ABB RobotStudio station: w7.rspag

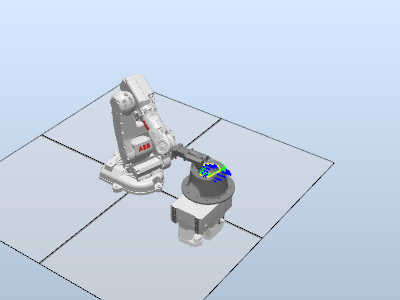
--- station ---
Station Project1 (saved by RobotStudio 22.3.10098.0)
Controller Controller1
  mechanical unit ROB_1: IRB140_6_81_C_03, 6 joints, base frame (0, 0, 0) mm
  mechanical unit M7DM1: MTD_250_M2009_REV1_01, 1 joints, base frame (584.98, -18.75, 250) mm, rotated rx 0 ry 0 rz 90 deg
Layout (positions relative to the parent item):
  - IRB140_6_81_C_03 [mechanism, from Robots\IRB140_6_81_C_G_03.rslib] at (0, 0, 0) mm; joint values [-0.3011, -0.1554, 0.7255, -0.5959, -0.6591, 0.4921] (rad or m)
  - MTD_250_M2009_REV1_01 [mechanism] at (584.98, -18.75, 250) mm, rotated rx 0 ry 0 rz 90 deg; joint values [0.0497] (rad or m)
      links: Base, Link1
  - gripped_pen [mechanism, from Components\gripped_pen.rslib] at (384.06, -95.88, 502.57) mm, rotated rx 0 ry 90 rz 2.85 deg
  - potty1 [part] at (690.16, 154.88, 241.77) mm, rotated rx 90 ry 0 rz 2.85 deg, size 275.1 x 194.8 x 257.3 mm
Attachment: gripped_pen is attached to IRB140_6_81_C_03 / Link6
Attachment: potty1 is attached to MTD_250_M2009_REV1_01 / Link1
Attachment: potty is attached to potty1

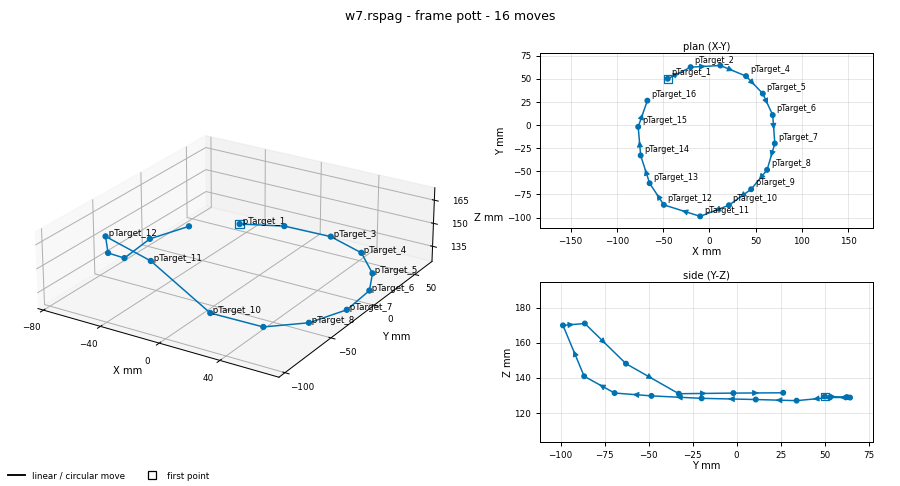
[picture p0: tool path of w7.rspag in frame pott, 16 of 16 moves have a stored position in this frame; points joined in program order, loops and branches not executed]
--- Controller Data/Controller1/RAPID/TASK1/PROGMOD/CalibData.mod ---
MODULE CalibData
    PERS tooldata gripped_pen:=[TRUE,[[121,0,178],[1,0,0,0]],[2,[0,50,88],[1,0,0,0],0,0,0]];
    PERS wobjdata pott:=[FALSE,FALSE,"M7DM1",[[0,0,0],[1,0,0,0]],[[0,0,0],[1,0,0,0]]];
    TASK PERS wobjdata potty:=[FALSE,TRUE,"",[[584.978108354,-18.746939063,250],[0.672758024,0,0,0.739862583]],[[0,0,0],[1,0,0,0]]];
    PERS wobjdata w3_2:=[FALSE,FALSE,"M7DM1",[[0,0,0],[1,0,0,0]],[[0,0,0],[1,0,0,0]]];
ENDMODULE

--- Controller Data/Controller1/RAPID/TASK1/PROGMOD/Gripper.mod ---
MODULE Gripper(READONLY)
    PROC Opengrippers()
        Reset closegripper;
        Set opengripper;
    ENDPROC

    PROC Closegrippers()
        Reset opengripper;
        Set closegripper;
    ENDPROC
ENDMODULE

--- Controller Data/Controller1/RAPID/TASK1/PROGMOD/Module1.mod ---
MODULE Module1
        CONST robtarget pTarget_1:=[[-45.03,50.16,129.476],[0.5,0.5,0.5,-0.5],[-1,-1,0,1],[1.561940022,9E+09,9E+09,9E+09,9E+09,9E+09]];
    CONST robtarget pTarget_2:=[[-20.282,62.744,129.127],[0.5,0.5,0.5,-0.5],[-1,-1,0,1],[3.28998974,9E+09,9E+09,9E+09,9E+09,9E+09]];
    CONST robtarget pTarget_3:=[[11.896,64.483,128.86],[0.5,0.5,0.5,-0.5],[-1,-1,0,1],[5.728209081,9E+09,9E+09,9E+09,9E+09,9E+09]];
    CONST robtarget pTarget_4:=[[39.689,53.042,128.927],[0.5,0.5,0.5,-0.5],[-1,-1,0,1],[8.105863915,9E+09,9E+09,9E+09,9E+09,9E+09]];
    CONST robtarget pTarget_5:=[[57.798,34.115,127.1],[0.5,0.5,0.5,-0.5],[-1,-1,0,1],[10.023360048,9E+09,9E+09,9E+09,9E+09,9E+09]];
    CONST robtarget pTarget_6:=[[68.525,10.908,127.738],[0.5,0.5,0.5,-0.5],[-1,-1,0,1],[11.363158759,9E+09,9E+09,9E+09,9E+09,9E+09]];
    CONST robtarget pTarget_7:=[[70.794,-19.857,128.419],[0.5,0.5,0.5,-0.5],[0,-1,0,1],[12.181392468,9E+09,9E+09,9E+09,9E+09,9E+09]];
    CONST robtarget pTarget_8:=[[62.436,-48.353,129.808],[0.5,0.5,0.5,-0.5],[0,-1,0,1],[11.998377809,9E+09,9E+09,9E+09,9E+09,9E+09]];
    CONST robtarget pTarget_9:=[[45.201,-69.327,131.428],[0.5,0.5,0.5,-0.5],[-1,-1,0,1],[10.863368437,9E+09,9E+09,9E+09,9E+09,9E+09]];
    CONST robtarget pTarget_10:=[[21.201,-86.605,140.96],[0.5,0.5,0.5,-0.5],[-1,-1,0,1],[8.564003859,9E+09,9E+09,9E+09,9E+09,9E+09]];
    CONST robtarget pTarget_11:=[[-9.927,-98.657,169.887],[0.5,0.5,0.5,-0.5],[-1,-1,0,1],[4.189417321,9E+09,9E+09,9E+09,9E+09,9E+09]];
    CONST robtarget pTarget_12:=[[-49.23,-86.236,170.954],[0.5,0.5,0.5,-0.5],[-1,-1,0,1],[1.111919617,9E+09,9E+09,9E+09,9E+09,9E+09]];
    CONST robtarget pTarget_13:=[[-64.618,-62.853,148.116],[0.5,0.5,0.5,-0.5],[-1,-1,0,1],[1.685696862,9E+09,9E+09,9E+09,9E+09,9E+09]];
    CONST robtarget pTarget_14:=[[-74.299,-32.791,131.037],[0.5,0.5,0.5,-0.5],[-1,-1,0,1],[2.190066988,9E+09,9E+09,9E+09,9E+09,9E+09]];
    CONST robtarget pTarget_15:=[[-76.984,-1.82,131.395],[0.5,0.5,0.5,-0.5],[-1,-1,0,1],[2.117495861,9E+09,9E+09,9E+09,9E+09,9E+09]];
    CONST robtarget pTarget_16:=[[-67.051,26.501,131.572],[0.5,0.5,0.5,-0.5],[-1,-1,0,1],[2.848945135,9E+09,9E+09,9E+09,9E+09,9E+09]];
!***********************************************************
    !
    ! Module:  Module1
    !
    ! Description:
    !   <Insert description here>
    !
    ! Author: sgmxu9
    !
    ! Version: 1.0
    !
    !***********************************************************


    !***********************************************************
    !
    ! Procedure main
    !
    !   This is the entry point of your program
    !
    !***********************************************************
    PROC main()
        !Add your code here
        Opengrippers;
        potty_top_1;
        Closegrippers;
    ENDPROC
    PROC potty_top_1()
        ActUnit M7DM1;
        MoveL pTarget_1,v1000,z100,gripped_pen\WObj:=pott;
        MoveL pTarget_2,v1000,z100,gripped_pen\WObj:=pott;
        MoveL pTarget_3,v1000,z100,gripped_pen\WObj:=pott;
        MoveL pTarget_4,v1000,z100,gripped_pen\WObj:=pott;
        MoveL pTarget_5,v1000,z100,gripped_pen\WObj:=pott;
        MoveL pTarget_6,v1000,z100,gripped_pen\WObj:=pott;
        MoveL pTarget_7,v1000,z100,gripped_pen\WObj:=pott;
        MoveL pTarget_8,v1000,z100,gripped_pen\WObj:=pott;
        MoveL pTarget_9,v1000,z100,gripped_pen\WObj:=pott;
        MoveL pTarget_10,v1000,z100,gripped_pen\WObj:=pott;
        MoveL pTarget_11,v1000,z100,gripped_pen\WObj:=pott;
        MoveL pTarget_12,v1000,z100,gripped_pen\WObj:=pott;
        MoveL pTarget_13,v1000,z100,gripped_pen\WObj:=pott;
        MoveL pTarget_14,v1000,z100,gripped_pen\WObj:=pott;
        MoveL pTarget_15,v1000,z100,gripped_pen\WObj:=pott;
        MoveL pTarget_16,v1000,z100,gripped_pen\WObj:=pott;
    ENDPROC
    PROC Path_10()
    ENDPROC
ENDMODULE

--- Controller Data/Controller1/SYSPAR/EIO.cfg ---
EIO:CFG_1.0:6:1::
#
INDUSTRIAL_NETWORK:

      -Name "DeviceNet" -Label "DeviceNet Master/Slave Network" -Address "2"
#
DEVICENET_DEVICE:

      -Name "board1" -VendorName "ABB Robotics" -ProductName "24 VDC I/O Device"\
      -Label "DSQC 652 24 VDC I/O Device" -ProductCode 26 -DeviceType 7\
      -ConnectionType "COS" -OutputSize 2 -InputSize 2
#
DEVICENET_INTERNAL_DEVICE:

      -Name "DN_Internal_Device" -VendorName "ABB Robotics"\
      -ProductName "DeviceNet Internal Slave Device"
#
EIO_SIGNAL:

      -Name "opengripper" -SignalType "DO" -Device "board1"\
      -Label "Open the Grippers" -DeviceMap "0" -Access "All"

      -Name "closegripper" -SignalType "DO" -Device "board1"\
      -Label "Close the Grippers" -DeviceMap "1" -Access "All"
